PROGRAM MAIN
VAR
	// TcUnit finds every FB_TestSuite instance by itself; it is enough to declare them here.
	fbEq2HorTests	: FB_EQ2HOR_Tests;
	fbHor2EqTests	: FB_HOR2EQ_Tests;
	fbCoRefractTests	: FB_CO_REFRACT_Tests;
	fbCoAberrationTests	: FB_CO_ABERRATION_Tests;
	fbCoNutateTests	: FB_CO_NUTATE_Tests;
END_VAR

TcUnit.RUN();

END_PROGRAM

(* stored: Version 1.1.0.1, ProductVersion 3.1.4024.15
   POU MAIN: Id {ffd4640f-010b-4811-97a9-18864652ad5b}, SpecialFunc None *)
